FUNCTION_BLOCK ParserTestFbt1
END_FUNCTION_BLOCK
